TYPE ST_SystemFileConfig :
STRUCT
	SchemaVersion : UDINT;
	ModuleCount : UINT;
	Modules : ARRAY[1..Param_Config.MaxTotalConfiguredModules] OF ST_ModuleFileConfig;
END_STRUCT
END_TYPE

(* stored: Version 1.1.0.1, ProductVersion 3.1.4026.18
   DUT ST_SystemFileConfig: Id {9aeab2a0-b447-4e97-903a-c039eb750d06} *)
